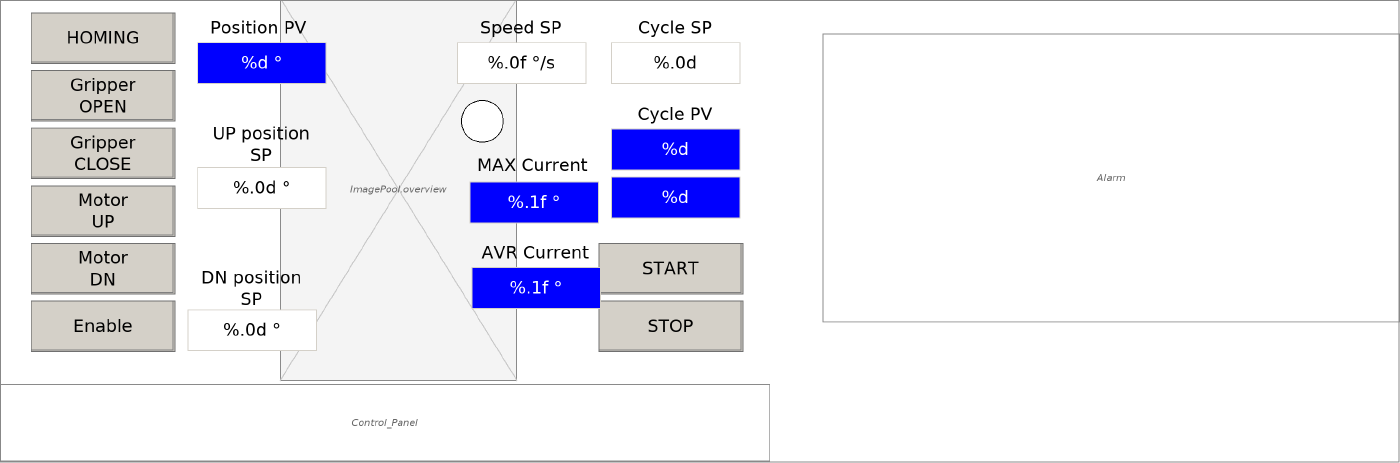
VISUALIZATION Overview  // 1455x482
    Button (32,13 150x53), "HOMING", colour toggle: GVL_IO.Homing_OK
        tap GVL_IO.Homing
    Button (32,73 150x53), "Gripper OPEN", colour toggle: GVL_IO.ixGripper_Unlock
        tap GVL_IO.Gripper_Open_cmd
    Button (32,133 150x53), "Gripper CLOSE", colour toggle: GVL_IO.TwoSensorLock
        tap GVL_IO.Gripper_Close_cmd
    Button (32,193 150x53), "Motor UP", colour toggle: GVL_IO.Motor_UP
        tap GVL_IO.Motor_UP
    Button (32,253 150x53), "Motor DN", colour toggle: GVL_IO.Motor_DN
        tap GVL_IO.Motor_DN
    Button (32,313 150x53), "Enable", colour toggle: GVL_IO.qxSTO_toDrive
        OnMouseClick: toggle GVL_IO.Enable_motor_cmd
    Frame (0,400 800x80)
        shows Control_Panel()
    Image (291,-2 246x398), image: ImagePool.overview
    Textfield (205,44 134x43), "%d °", text variable: GVL_IO.Position_PV_HMI
    Label (206,13 131x32), "Position PV"
    Label (206,125 131x50), "UP position SP"
    Textfield (205,174 134x43), "%.0d °", text variable: GVL_IO.Position_UP_SP
        OnMouseClick: write the text variable via Default
    Label (196,275 131x50), "DN position SP"
    Textfield (195,322 134x43), "%.0d °", text variable: GVL_IO.Position_DN_SP
        OnMouseClick: write the text variable via Default
    Label (636,13 131x32), "Cycle SP"
    Textfield (635,44 134x43), "%.0d", text variable: GVL_IO.Cycle_SP
        OnMouseClick: write the text variable via Default
    Textfield (475,44 134x43), "%.0f °/s", text variable: GVL_IO.Speed_SP
        OnMouseClick: write the text variable via Default
    Label (476,13 131x32), "Speed SP"
    Label (636,103 131x32), "Cycle PV"
    Textfield (635,134 134x43), "%d", text variable: GVL_IO.Cycle_PV
    Button (622,253 150x53), "START"
        tap GVL_IO.Start
    Button (622,313 150x53), "STOP", colour toggle: GVL_IO.Stop
        tap GVL_IO.Stop
    Textfield (635,184 134x43), "%d", text variable: ServoCtrl.Position
    Ellipse (479,104 44x44), colour toggle: GVL_IO.ixHome_Position
    Label (488,156 131x32), "MAX Current"
    Textfield (488,189 134x43), "%.1f °", text variable: GVL_IO.Motor_I_MAX
    Label (491,247 131x32), "AVR Current"
    Textfield (490,278 134x43), "%.1f °", text variable: GVL_IO.Motor_I_AVR
    Frame (855,35 600x300), invisible if: GVL_IO.Error = 0
        shows Alarm()
        p3560616238: -750
END_VISUALIZATION

(* stored: Version 1.1.0.1, ProductVersion 3.1.4024.15
   Visu Overview: Id {c8af26be-14f3-46be-b772-5a548960db44} *)
